TYPE ST_PistonRange :
STRUCT
END_STRUCT
END_TYPE

(* stored: Version 1.1.0.1, ProductVersion 3.1.4024.10
   DUT ST_PistonRange: Id {8b317ca5-9e1d-4164-abfc-6c7090e6899c} *)
